TYPE IoChuckPhotoLum :
STRUCT		
	OutputVaccum100mm  AT %Q* : BOOL;
	OutputVaccum150mm AT %Q* : BOOL;		
	OutputVaccum200mm AT %Q* :BOOL;		
END_STRUCT
END_TYPE

(* stored: Version 1.1.0.1, ProductVersion 3.1.4024.12
   DUT IoChuckPhotoLum: Id {d09c5408-7883-4f49-92d2-74e6234334cd} *)
